{attribute 'GeneratedUsingTerminal: EL6201-0000-0017'}
{attribute addProperty BoxType "EL6201-0000-0017"}
{attribute addProperty Id "Slave_3A_DO0BOOL1Slave_3A_DO1BOOL1Slave_3A_DO2BOOL1Slave_3A_DO3BOOL1Slave_3B_DO0BOOL1Slave_3B_DO1BOOL1Slave_3B_DO2BOOL1Slave_3B_DO3BOOL1"}
{attribute addProperty CRC "935275816"}
{attribute addProperty Size "8"}
TYPE Slave_3_Outputs_37BF2D28 :
STRUCT
	{attribute addProperty Name "Slave_3A_DO0"}
	Slave_3A_DO0 : BOOL;
	{attribute addProperty Name "Slave_3A_DO1"}
	Slave_3A_DO1 : BOOL;
	{attribute addProperty Name "Slave_3A_DO2"}
	Slave_3A_DO2 : BOOL;
	{attribute addProperty Name "Slave_3A_DO3"}
	Slave_3A_DO3 : BOOL;
	{attribute addProperty Name "Slave_3B_DO0"}
	Slave_3B_DO0 : BOOL;
	{attribute addProperty Name "Slave_3B_DO1"}
	Slave_3B_DO1 : BOOL;
	{attribute addProperty Name "Slave_3B_DO2"}
	Slave_3B_DO2 : BOOL;
	{attribute addProperty Name "Slave_3B_DO3"}
	Slave_3B_DO3 : BOOL;
END_STRUCT
END_TYPE

(* stored: Version 1.2.0.0, ProductVersion 3.1.4024.9
   DUT Slave_3_Outputs_37BF2D28: Id {7f3989c9-2786-4fee-af31-ac9dcf69ed51} *)
